{attribute 'qualified_only'}
{attribute 'strict'}
TYPE E_LED :
(
	MaintenanceBtn := 0,
	AbortFlowBtn,
	DoorUnlockBtn,
	Aarm
);
END_TYPE

(* stored: Version 1.1.0.1, ProductVersion 3.1.4022.12
   DUT E_LED: Id {bb63c7ef-1cce-4133-987f-6b42ccaa7405} *)
